# EPICS StreamDevice protocol: dma4500mSup/dma4500m.proto
# Stream Device Protocol for the Anton Paar DMA 4500 M
# Density Meter.
#
# Andreas Hagelberg
# European Spallation Source ERIC
# March 2018

replytimeout = 5000;
readtimeout  = 5000;
terminator = CR;

# Make sure stream buffer is empty
@init { out " " }

set_temperature { out "settemperature %.2f"; } # in "%{accepted|wrong parameter value|not allowed during measurement}"; }
start { out "start"; in "%{measurement already started|measurement started}" }
abort { out "abort"; in "measurement %{aborted|not started}" }
finished { out "finished"; in "measurement %{not started|not finished|finished}" }
data { out "getdata"; in "%{data: %f;%f;%f;%s|no new data available}" }
units { out "getdataunit"; in "data unit: %s" }
serial { out "getid"; in "serial number: %s" }
method { out "getmethodname"; in "method name: %s" }
legend { out "getdatahead"; in "data head: %s" }

density_unit {
  out "getdataunit";
  in "data unit: %[^;];%*[^;];%*[^;];%*s";
}

temp_unit {
  in "data unit: %*[^;];%*[^;];%[^;];%*s";
}

get_data_density_only {
  out "getdata";
  in "data: %(\$1)f;%(\$2)f;%(\$3)s";
}

get_temperature_setpoint {
  out "getrawdata";
  in "%*f;%*f;%f;%*s";
}
